SUBAPPLICATION Maehwerksklappung_IXA (* Mähwerksklappung Aufgabe Febr. 2026 *)
  (* Standard: 61499-2 *)
  (* Version 1.0, 2026-02-23, Herr Lehrer *)
  PACKAGE Meins;
  IMPORT logiBUS::io::DI::logiBUS_DI::Input_I1;
  IMPORT logiBUS::io::DI::logiBUS_DI::Input_I2;
  IMPORT logiBUS::io::DI::logiBUS_DI::Input_I3;
  IMPORT logiBUS::io::DI::logiBUS_DI::Input_I4;
  IMPORT logiBUS::io::DI::logiBUS_DI::Input_I5;
  IMPORT logiBUS::io::DI::logiBUS_DI::Input_I6;
  IMPORT logiBUS::io::DQ::logiBUS_DO::Output_Q1;
  IMPORT logiBUS::io::DQ::logiBUS_DO::Output_Q2;
  IMPORT logiBUS::io::DQ::logiBUS_DO::Output_Q3;
  IMPORT logiBUS::io::DQ::logiBUS_DO::Output_Q4;
  IMPORT logiBUS::io::DQ::logiBUS_DO::Output_Q5;
  IMPORT logiBUS::io::DQ::logiBUS_DO::Output_Q6;
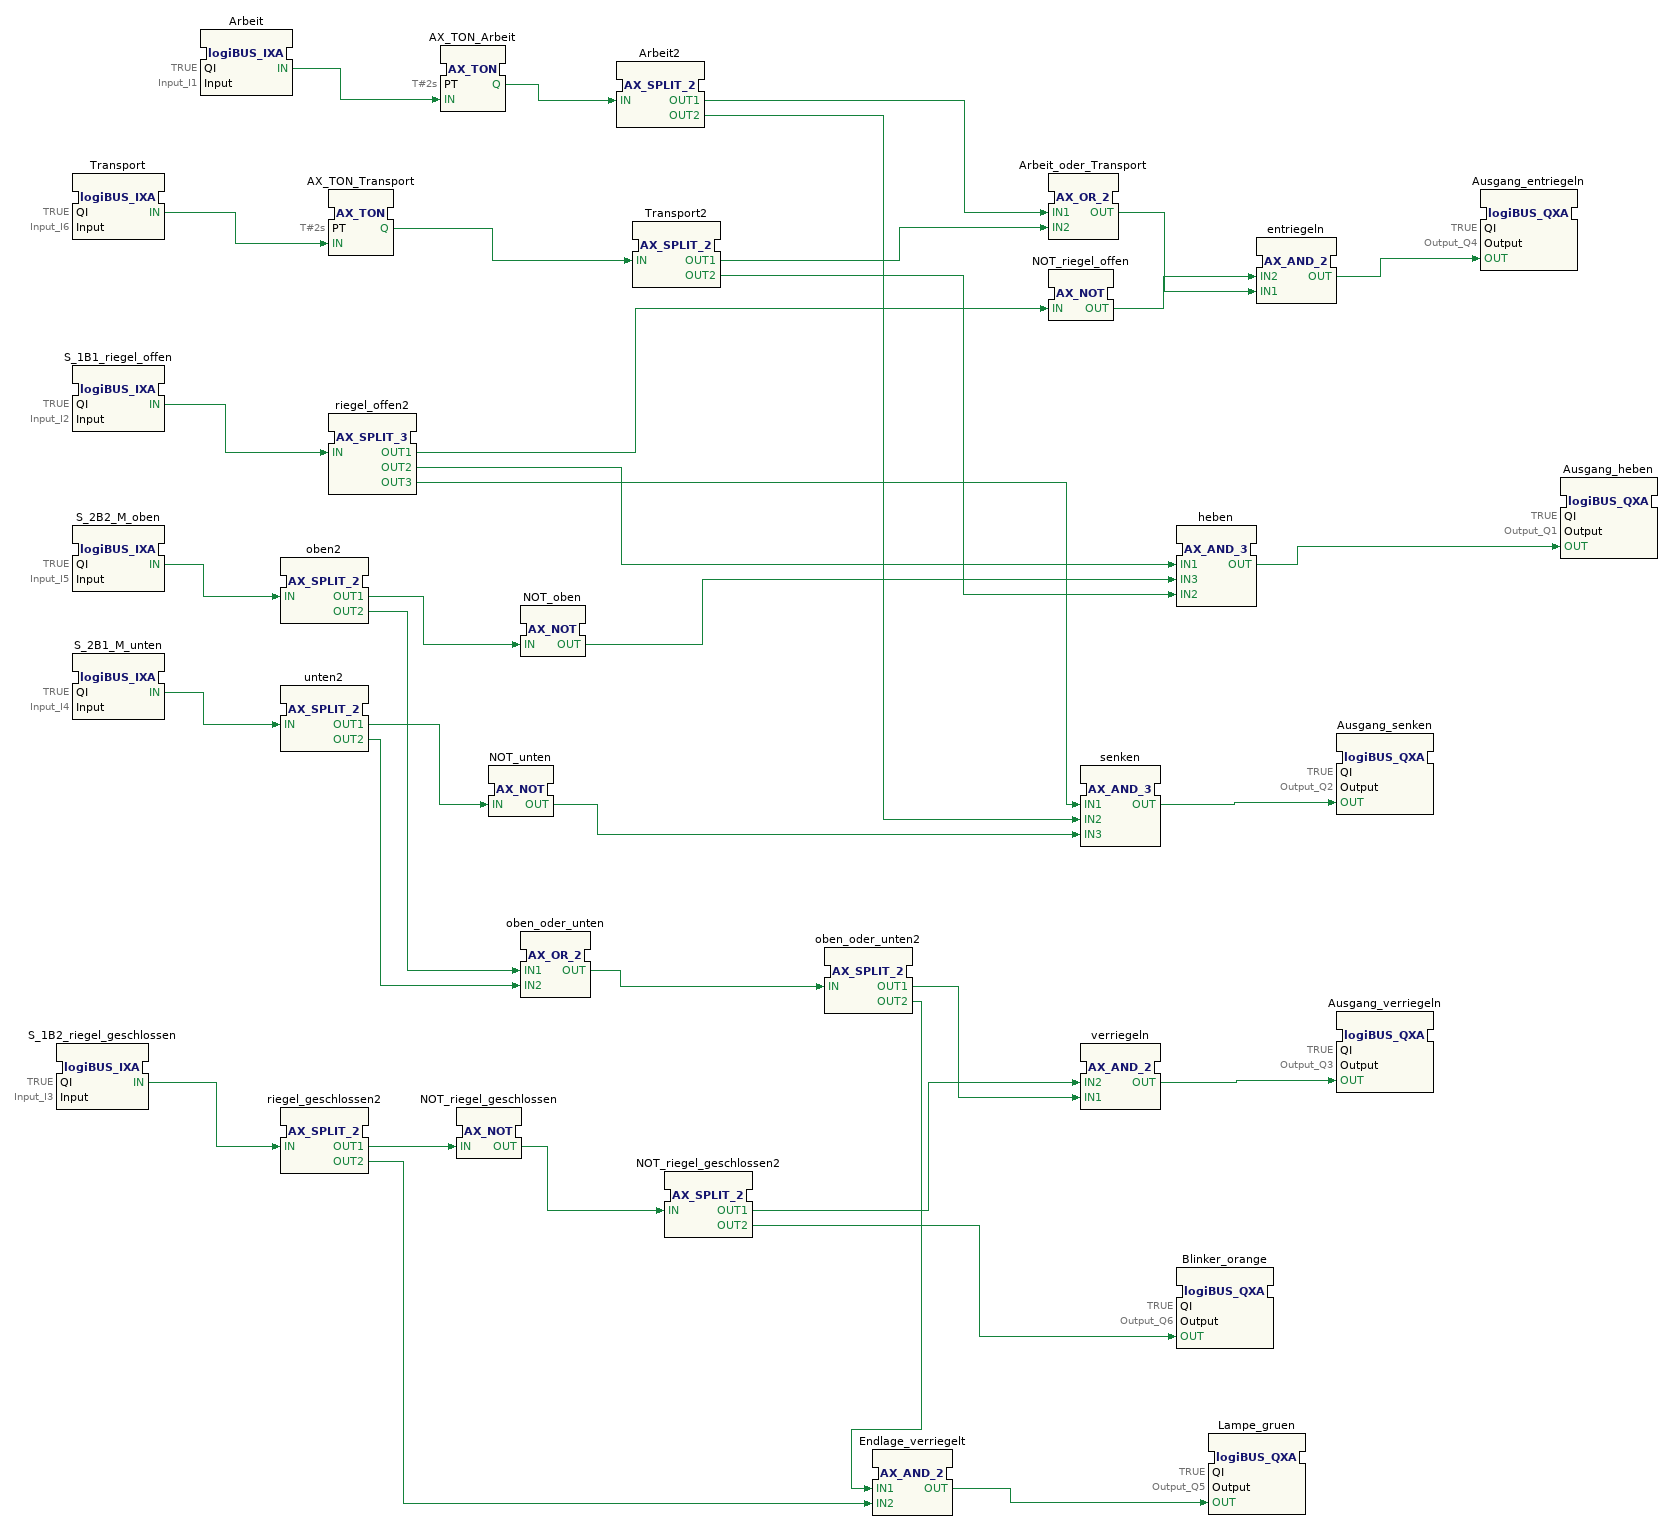
  (* UNTEN *)
  (* A. Entriegeln (Bolzen fährt ein) Damit das Mähwerk überhaupt fahren darf, muss bei Tastendruck zuerst der Riegel öffnen.Logik: Y_1 = (S_1 or S_2) and not 1B1 Erklärung: Wenn der Taster "Transport" (S_1) oder "Arbeit" (S_2) gedrückt wird UND der Riegel noch nicht in der Position "Offen" ist (1B1) , wird der Ausgang "Riegel öffnen" (Y_1)  angesteuert. *)
  (* Heben (Transport): Y_3 = S_1 and 1B1 and not 2B2 Erklärung: Der Ausgang "Mähwerk heben" (Y_3) ist nur aktiv, solange S_1 gedrückt bleibt, der Riegel "Offen" meldet (1B1) und die obere Endlage (2B2) noch nicht erreicht ist. Lässt der Fahrer S_1 los, wird die Bedingung falsch, Y_3 fällt ab und das 5/3-Wegeventil stoppt den Zylinder sofort. *)
  (* Senken (Arbeit): Y_4 = S_2 and 1B1 and not 2B1 Erklärung: Analog zum Heben. Der Ausgang "Mähwerk senken" (Y_4) ist nur aktiv, solange S_2 gedrückt ist, der Riegel offen ist und die untere Endlage (2B1) nicht erreicht ist. *)
  (* Logik: Y_2 = (2B2 or 2B1) and not 1B2 Erklärung: Sobald das Mähwerk ganz oben (2B2) oder ganz unten (2B1) ist UND der Riegel noch nicht zu ist (not 1B2) , wird der Ausgang "Riegel schließen" (Y_2) aktiviert. *)
  (* Warnleuchte (H_1): Soll während des gesamten Bewegungsablaufs leuchten/blinken. Das ist der Fall, solange der Riegel nicht komplett geschlossen ist. H_1 = not 1B2 *)
  (* Statusleuchte (H_2): Signalisert den sicheren Zustand (Verriegelt in Endlage).H_2 = 1B2 and (2B2 or 2B1) *)
  FBS
    Ausgang_heben : logiBUS::io::DQ::logiBUS_QXA(QI := TRUE, Output := Output_Q1);
    Ausgang_senken : logiBUS::io::DQ::logiBUS_QXA(QI := TRUE (* Event Input Qualifier *), Output := Output_Q2);
    Ausgang_entriegeln : logiBUS::io::DQ::logiBUS_QXA(QI := TRUE, Output := Output_Q4);
    Ausgang_verriegeln : logiBUS::io::DQ::logiBUS_QXA(QI := TRUE, Output := Output_Q3);
    Lampe_gruen : logiBUS::io::DQ::logiBUS_QXA(QI := TRUE, Output := Output_Q5);
    Blinker_orange : logiBUS::io::DQ::logiBUS_QXA(QI := TRUE, Output := Output_Q6);
    Arbeit : logiBUS::io::DI::logiBUS_IXA(QI := TRUE, Input := Input_I1);
    S_1B1_riegel_offen : logiBUS::io::DI::logiBUS_IXA(QI := TRUE, Input := Input_I2);
    S_1B2_riegel_geschlossen : logiBUS::io::DI::logiBUS_IXA(QI := TRUE, Input := Input_I3);
    S_2B2_M_oben : logiBUS::io::DI::logiBUS_IXA(QI := TRUE, Input := Input_I5);
    S_2B1_M_unten : logiBUS::io::DI::logiBUS_IXA(QI := TRUE, Input := Input_I4);
    Transport : logiBUS::io::DI::logiBUS_IXA(QI := TRUE, Input := Input_I6);
    AX_TON_Arbeit : adapter::events::unidirectional::timers::AX_TON(PT := T#2s);
    AX_TON_Transport : adapter::events::unidirectional::timers::AX_TON(PT := T#2s);
    NOT_riegel_offen : adapter::booleanOperators::AX_NOT;
    entriegeln : adapter::booleanOperators::AX_AND_2;
    Arbeit_oder_Transport : adapter::booleanOperators::AX_OR_2;
    riegel_offen2 : adapter::events::unidirectional::AX_SPLIT_3;
    heben : adapter::booleanOperators::AX_AND_3;
    NOT_oben : adapter::booleanOperators::AX_NOT;
    senken : adapter::booleanOperators::AX_AND_3;
    Arbeit2 : adapter::events::unidirectional::AX_SPLIT_2;
    NOT_unten : adapter::booleanOperators::AX_NOT;
    verriegeln : adapter::booleanOperators::AX_AND_2;
    NOT_riegel_geschlossen : adapter::booleanOperators::AX_NOT;
    oben_oder_unten : adapter::booleanOperators::AX_OR_2;
    oben2 : adapter::events::unidirectional::AX_SPLIT_2;
    unten2 : adapter::events::unidirectional::AX_SPLIT_2;
    NOT_riegel_geschlossen2 : adapter::events::unidirectional::AX_SPLIT_2;
    oben_oder_unten2 : adapter::events::unidirectional::AX_SPLIT_2;
    Endlage_verriegelt : adapter::booleanOperators::AX_AND_2;
    riegel_geschlossen2 : adapter::events::unidirectional::AX_SPLIT_2;
    Transport2 : adapter::events::unidirectional::AX_SPLIT_2;
  END_FBS
  ADAPTER_CONNECTIONS
    Arbeit.IN TO AX_TON_Arbeit.IN;
    riegel_offen2.OUT1 TO NOT_riegel_offen.IN;
    NOT_riegel_offen.OUT TO entriegeln.IN2;
    Arbeit_oder_Transport.OUT TO entriegeln.IN1;
    entriegeln.OUT TO Ausgang_entriegeln.OUT;
    Arbeit2.OUT1 TO Arbeit_oder_Transport.IN1;
    heben.OUT TO Ausgang_heben.OUT;
    S_1B1_riegel_offen.IN TO riegel_offen2.IN;
    oben2.OUT1 TO NOT_oben.IN;
    riegel_offen2.OUT2 TO heben.IN1;
    NOT_oben.OUT TO heben.IN3;
    senken.OUT TO Ausgang_senken.OUT;
    riegel_offen2.OUT3 TO senken.IN1;
    AX_TON_Arbeit.Q TO Arbeit2.IN;
    Arbeit2.OUT2 TO senken.IN2;
    unten2.OUT1 TO NOT_unten.IN;
    NOT_unten.OUT TO senken.IN3;
    verriegeln.OUT TO Ausgang_verriegeln.OUT;
    NOT_riegel_geschlossen2.OUT1 TO verriegeln.IN2;
    oben_oder_unten2.OUT1 TO verriegeln.IN1;
    S_2B2_M_oben.IN TO oben2.IN;
    S_2B1_M_unten.IN TO unten2.IN;
    oben2.OUT2 TO oben_oder_unten.IN1;
    unten2.OUT2 TO oben_oder_unten.IN2;
    NOT_riegel_geschlossen.OUT TO NOT_riegel_geschlossen2.IN;
    NOT_riegel_geschlossen2.OUT2 TO Blinker_orange.OUT;
    oben_oder_unten.OUT TO oben_oder_unten2.IN;
    Endlage_verriegelt.OUT TO Lampe_gruen.OUT;
    oben_oder_unten2.OUT2 TO Endlage_verriegelt.IN1;
    S_1B2_riegel_geschlossen.IN TO riegel_geschlossen2.IN;
    riegel_geschlossen2.OUT1 TO NOT_riegel_geschlossen.IN;
    riegel_geschlossen2.OUT2 TO Endlage_verriegelt.IN2;
    Transport.IN TO AX_TON_Transport.IN;
    AX_TON_Transport.Q TO Transport2.IN;
    Transport2.OUT1 TO Arbeit_oder_Transport.IN2;
    Transport2.OUT2 TO heben.IN2;
  END_CONNECTIONS
END_SUBAPPLICATION
